RoboDK station: scrab_master.rdk

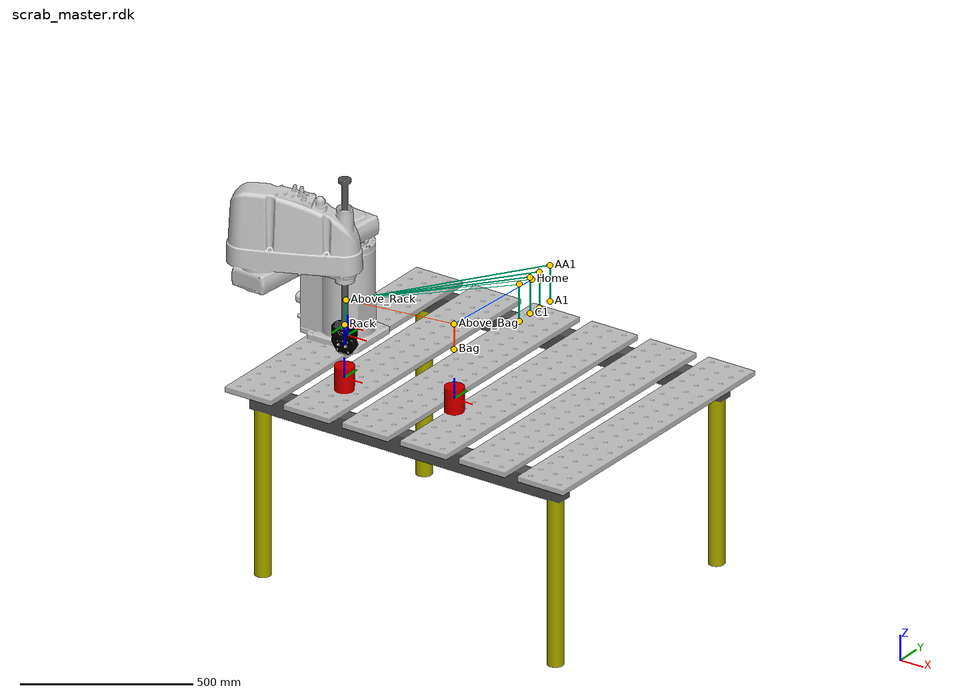
[picture v0: the station drawn from its stored meshes, robots at their saved joint values, targets as dots, program paths as lines]
Station scrab_master. Poses are relative to the parent item; angles as X-Y-Z fixed-axis rotations.
  - frame Motoman MYS650L Base at (0, 0, 0) mm
    - robot Motoman MYS650L: 4 axes, payload 6 kg, reach 650 mm, repeatability 0.02 mm, weight 28 kg
        modified DH rows (alpha deg, a mm, theta deg, d mm): 0, 0, 0, 0; 0, 400, 0, 0; 0, 250, 0, 31 linear; 180, 0, 0, 0
        joint limits [-160, -140, 0, -360] to [160, 140, 330, 360]; home [0, 0, 330, 0]; saved at [-94.602, 117.866, 177.358, 23.264]
      - robot RobotiQ 2F85: 1 axes, payload 5 kg
          joint limits [0] to [85]; home [85]; saved at [85]
        - frame Grip at (0, 0, 0) mm
          - target Open (Cartesian target) at (0, 0, 0) mm; joints [85] of RobotiQ 2F85
          - target Pick (Cartesian target) at (0, 0, 0) mm; joints [60] of RobotiQ 2F85
    - object Table at (500, 0, 0) mm, size 1193.8 x 965.2 x 609.6 mm, geometry from welding_table.sld
    - target Home (Cartesian target) at (650, 0, 361) mm, rotated rx 180 ry 0 rz 0 deg; joints [0, 0, 330, 0] of Motoman MYS650L
    - target Above_Bag (Cartesian target) at (549.35, -249.89, 289.38) mm, rotated rx 180 ry 0 rz 0 deg; joints [-41.454, 44.875, 258.385, 3.421] of Motoman MYS650L
    - target Bag (Cartesian target) at (549.35, -249.89, 208.3) mm, rotated rx 180 ry 0 rz 0 deg; joints [-41.454, 44.875, 177.296, 3.421] of Motoman MYS650L
    - target Above_Rack (Cartesian target) at (203.14, -299.97, 289.38) mm, rotated rx 180 ry 0 rz 0 deg; joints [-93.777, 117.146, 258.385, 23.369] of Motoman MYS650L
    - target Rack (Cartesian target) at (197.58, -299.97, 208.36) mm, rotated rx 180 ry 0 rz 0 deg; joints [-94.602, 117.866, 177.358, 23.264] of Motoman MYS650L
    - target A1 (Cartesian target) at (559.43, 219.74, 178.23) mm, rotated rx 180 ry 0 rz 0 deg; joints [4.012, 46.075, 147.227, 50.087] of Motoman MYS650L
    - target AA1 (Cartesian target) at (559.43, 219.74, 294.41) mm, rotated rx 180 ry 0 rz 0 deg; joints [4.012, 46.075, 263.414, 50.087] of Motoman MYS650L
    - target B1 (Cartesian target) at (559.43, 166.81, 178.23) mm, rotated rx 180 ry 0 rz 0 deg; joints [-3.599, 53.743, 147.227, 50.144] of Motoman MYS650L
    - target AB1 (Cartesian target) at (559.43, 166.81, 293.43) mm, rotated rx 180 ry 0 rz 0 deg; joints [-3.599, 53.743, 262.434, 50.144] of Motoman MYS650L
    - target C1 (Cartesian target) at (559.43, 118.94, 178.23) mm, rotated rx 180 ry 0 rz 0 deg; joints [-9.871, 58.465, 147.227, 48.594] of Motoman MYS650L
    - target AC1 (Cartesian target) at (559.43, 118.94, 295.45) mm, rotated rx 180 ry 0 rz 0 deg; joints [-9.871, 58.465, 264.454, 48.594] of Motoman MYS650L
    - target AD1 (Cartesian target) at (559.43, 63.9, 295.45) mm, rotated rx 180 ry 0 rz 0 deg; joints [-16.517, 61.79, 264.454, 45.273] of Motoman MYS650L
    - target D1 (Cartesian target) at (559.43, 63.9, 174.88) mm, rotated rx 180 ry 0 rz 0 deg; joints [-16.517, 61.79, 143.883, 45.273] of Motoman MYS650L
  - frame Rack at (197.02, -300, 38.84) mm
    - object Part at (0, 0, 0) mm, size 60 x 60 x 80 mm, geometry from part.sld
  - frame Bag at (550, -250, 50) mm
    - object Part at (0, 0, 0) mm, size 60 x 60 x 80 mm, geometry from part.sld
  - program Pick (1 instructions, listed below)
  - program Place (1 instructions, listed below)
  - program Robar1 (10 instructions, listed below)
  - program Robar2 (9 instructions, listed below)
  - program PlaceA (34 instructions, listed below)
  - program Main (6 instructions, listed below)
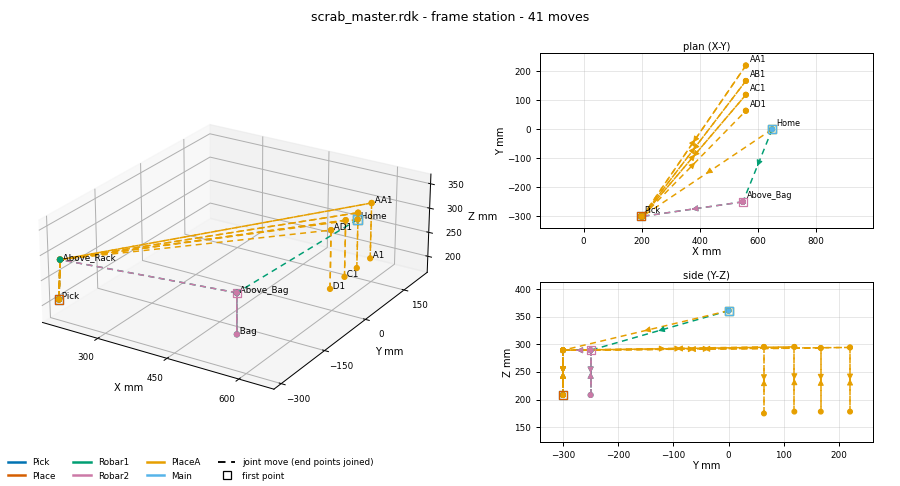
[picture p0: tool path of scrab_master.rdk in frame station, 41 of 41 moves have a stored position in this frame; points joined in program order, loops and branches not executed]

--- program Pick (robot RobotiQ 2F85) ---
  MoveJ (Pick)

--- program Place (robot RobotiQ 2F85) ---
  MoveJ (Open)

--- program Robar1 (robot Motoman MYS650L) ---
  Est. Ref.: Motoman MYS650L Base
  MoveJ (Home)
  MoveJ (Above_Bag)
  MoveJ (Bag)
  Llamar Pick
  MoveJ (Above_Bag)
  MoveJ (Above_Rack)
  MoveJ (Rack)
  Llamar Place
  MoveJ (Above_Rack)

--- program Robar2 (robot Motoman MYS650L) ---
  Est. Ref.: Motoman MYS650L Base
  MoveJ (Above_Bag)
  MoveJ (Bag)
  Llamar Pick
  MoveJ (Above_Bag)
  MoveJ (Above_Rack)
  MoveJ (Rack)
  Llamar Place
  MoveJ (Above_Rack)

--- program PlaceA (robot Motoman MYS650L) ---
  Est. Ref.: Motoman MYS650L Base
  MoveJ (Home)
  MoveJ (Above_Rack)
  MoveJ (Rack)
  Llamar Pick
  MoveJ (Above_Rack)
  MoveJ (AA1)
  MoveJ (A1)
  Llamar Place
  MoveJ (AA1)
  MoveJ (Above_Rack)
  MoveJ (Rack)
  Llamar Pick
  MoveJ (Above_Rack)
  MoveJ (AB1)
  MoveJ (B1)
  Llamar Place
  MoveJ (AB1)
  MoveJ (Above_Rack)
  MoveJ (Rack)
  Llamar Pick
  MoveJ (Above_Rack)
  MoveJ (AC1)
  MoveJ (C1)
  Llamar Place
  MoveJ (AC1)
  MoveJ (Above_Rack)
  MoveJ (Rack)
  Llamar Pick
  MoveJ (Above_Rack)
  MoveJ (AD1)
  MoveJ (D1)
  Llamar Place
  MoveJ (AD1)

--- program Main (robot Motoman MYS650L) ---
  Llamar PlaceA
  Llamar Robar1
  Llamar Robar2
  Llamar Robar2
  Llamar Robar2
  MoveJ (Home)
